KUKA KRL data list: Glode_HanGao.dat

&ACCESS RVO1
&REL 506
&PARAM EDITMASK = *
&PARAM TEMPLATE = C:\KRC\Roboter\Template\vorgabe
&PARAM DISKPATH = KRC:\R1\Program\HG
DEFDAT  GLODE_HANGAO PUBLIC



GLOBAL BOOL EKI_Server_Ini=TRUE
GLOBAL BOOL EKI_Server_Open=TRUE
GLOBAL BOOL EKI_Server_Connect=TRUE
GLOBAL BOOL EKI_Server_Receive=FALSE
GLOBAL BOOL EKI_Server_Send=FALSE
GLOBAL BOOL EKI_Server_Reset=FALSE


;--------DECL_Enum---------------
GLOBAL ENUM Sink_Type_Enum UpDown_One,LeftRight_One,LeftRight_Two,Null
GLOBAL ENUM Area_Enum L0,C45,L90,C135,L180,C225,L270,C315,N45,N135,N225,N315
GLOBAL ENUM Pos_Type_Enum C_LIN_POS,C_CIR_POS,L_LIN_POS
GLOBAL ENUM Work_Area_Enum A0,A90,A270
GLOBAL ENUM Vision_Model_Enum Calibration,Find_Model
GLOBAL ENUM Vision_Type_Enum Vision_Run,Vision_No,Vision_Text
GLOBAL ENUM Vision_PATH_Enum X,Y,Z,XY,XZ,YZ,XYZ,XYZABC
;----------------------------------
;---DECL-STRUC-------------------------


GLOBAL STRUC Surround_Welding_Type BOOL Write_Status,REAL Sink_Size_Long,REAL Sink_Size_Width,REAL Sink_Size_R,REAL Sink_Size_Short_Side,REAL Sink_Size_Short_OnePos,REAL Sink_Size_Short_TwoPos,REAL Sink_Size_Pots_Thick,REAL Sink_Size_Panel_Thick,INT Sink_Model,REAL Sink_Size_Left_Distance,REAL Sink_Size_Down_Distance,Sink_Type_Enum Sink_Type
GLOBAL STRUC LSC_TOOL_TYP INT LSR_MAX_PWR,INT LSR_MIN_PWR,INT LSR_Prg,REAL SNSR_Prg,INT SNSR_State,REAL GAS_Pressure,INT LSR_Dly,INT GAS_Pre_Flow,INT GAS_Post_Flow
GLOBAL STRUC Offset_POS REAL X,REAL Y,REAL Z,REAL A,REAL B,REAL C
GLOBAL STRUC Offset_CIR REAL C_X,REAL C_Y,REAL C_Z,REAL C_A,REAL C_B,REAL C_C
GLOBAL STRUC Calculate_Lin_Const REAL A,REAL B,REAL C
GLOBAL STRUC Calibration_Sink_TYP REAL Long,REAL Width
GLOBAL STRUC Calibrate_Data BOOL Calibrate_State,INT Plan_Base_No,CHAR Calib_Pos_Name_1[20],CHAR Calib_Pos_Name_2[20],CHAR Calib_Pos_Name_3[20],CHAR Calib_Pos_Name_4[20],CHAR Calib_Pos_Name_5[20],CHAR Calib_Pos_Name_6[20],CHAR Calib_Pos_Name_7[20],CHAR Calib_Pos_Name_8[20],CHAR Calib_Pos_Name_9[20],CHAR Calib_Pos_Name_10[20]



GLOBAL STRUC Surr_Welding_Craft_Type CHAR Welding_Name[20],E6POS Welding_Pos,REAL Welding_Power,REAL Welding_Speed,REAL Welding_Angle,INT Welding_CDIS,INT Welding_ACC,Offset_POS Welding_Offset,Offset_CIR Welding_Offset_CIR



;-------------------------------------


;----------DECL_Value----------------------
DECL GLOBAL Surround_Welding_Type SW_DEFAULT={Sink_Size_Long 50.0000,Sink_Size_Width 345.000,Sink_Size_R 10.0000,Sink_Size_Pots_Thick 0.750000,Sink_Size_Panel_Thick 2.85000,Sink_Model 952154,Sink_Type #UpDown_One}
DECL GLOBAL LSC_TOOL_TYP LTDEFAULT={LSR_MAX_PWR 500,LSR_MIN_PWR 50,LSR_Prg 1,SNSR_Prg 1.00000,SNSR_State 0,GAS_Pressure 1.00000,LSR_Dly 100,GAS_Pre_Flow 0,GAS_Post_Flow 0}
DECL GLOBAL Offset_POS FFDEFAULT={X 0.0,Y 0.0,Z 0.0,A 0.0,B 0.0,C 0.0}
DECL GLOBAL Offset_CIR FCDEFAULT={C_X 0.0,C_Y 0.0,C_Z 0.0,C_A 0.0,C_B 0.0,C_C 0.0}
DECL GLOBAL Calibrate_Data CDDEFAULT={Calibrate_State FALSE,Plan_Base_No 5,Calib_Pos_Name_1[] " ",Calib_Pos_Name_2[] " ",Calib_Pos_Name_3[] " ",Calib_Pos_Name_4[] " ",Calib_Pos_Name_5[] " ",Calib_Pos_Name_6[] " ",Calib_Pos_Name_7[] " ",Calib_Pos_Name_8[] " ",Calib_Pos_Name_9[] " ",Calib_Pos_Name_10[] " "}
DECL GLOBAL E6POS PODEFAULT={X 0.0,Y 0.0,Z 0.0,A 0.0,B 0.0,C 0.0}
DECL GLOBAL E6POS XDEFAULT={X 0.0,Y 0.0,Z 0.0,A 0.0,B 0.0,C 0.0,S 2,T 2,E1 0.0,E2 0.0,E3 0.0,E4 0.0,E5 0.0,E6 0.0}



DECL GLOBAL Surround_Welding_Type Camera_Calibration_Data={Sink_Size_Long 632.000,Sink_Size_Width 352.000,Sink_Size_R 10.0000,Sink_Size_Short_Side 23.0000,Sink_Size_Short_OnePos 36.0000,Sink_Size_Short_TwoPos 328.000,Sink_Size_Pots_Thick 0.0,Sink_Size_Panel_Thick 0.0,Sink_Model 952154,Sink_Size_Left_Distance 24.0000,Sink_Size_Down_Distance 24.0000,Sink_Type #LeftRight_One}

DECL GLOBAL E6POS N1_Cam_45_POS={X 293.000,Y 90.0000,Z -80.0000,A 0.0,B 0.0,C 0.0,S 2,T 10,E1 0.0,E2 0.0,E3 0.0,E4 0.0,E5 0.0,E6 0.0}
DECL GLOBAL E6POS N1_Cam_135_POS={X -42.0000,Y 90.0000,Z -80.0000,A 0.0,B 0.0,C 0.0,S 2,T 10,E1 0.0,E2 0.0,E3 0.0,E4 0.0,E5 0.0,E6 0.0}
DECL GLOBAL E6POS N1_Cam_225_POS={X -40.0000,Y 716.000,Z -80.0000,A 0.0,B 0.0,C 0.0,S 2,T 43,E1 0.0,E2 0.0,E3 0.0,E4 0.0,E5 0.0,E6 0.0}
DECL GLOBAL E6POS N1_Cam_315_POS={X 295.000,Y 714.000,Z -80.0000,A 0.0,B 0.0,C 0.0,S 2,T 43,E1 0.0,E2 0.0,E3 0.0,E4 0.0,E5 0.0,E6 0.0}

DECL GLOBAL E6POS N2_Cam_45_POS={X 293.122131,Y 89.9176636,Z -80.0293961,A 0.0,B 0.0,C 0.0,S 2,T 10,E1 0.0,E2 0.0,E3 0.0,E4 0.0,E5 0.0,E6 0.0}
DECL GLOBAL E6POS N2_Cam_135_POS={X -42.3839874,Y 91.8151550,Z -80.0254822,A 0.0,B 0.0,C 0.0,S 2,T 10,E1 0.0,E2 0.0,E3 0.0,E4 0.0,E5 0.0,E6 0.0}
DECL GLOBAL E6POS N2_Cam_225_POS={X -39.7999954,Y 716.082336,Z -80.0293350,A 0.0,B 0.0,C 0.0,S 2,T 43,E1 0.0,E2 0.0,E3 0.0,E4 0.0,E5 0.0,E6 0.0}
DECL GLOBAL E6POS N2_Cam_315_POS={X 294.984924,Y 714.198059,Z -80.0293350,A 0.0,B 0.0,C 0.0,S 2,T 43,E1 0.0,E2 0.0,E3 0.0,E4 0.0,E5 0.0,E6 0.0}

DECL GLOBAL E6POS N45_OFFSET_POS={X 375.888,Y 19.1080,Z 0.0,A 0.0,B 0.0,C 0.0}
DECL GLOBAL E6POS N135_OFFSET_POS={X 19.2480,Y 19.4280,Z 0.0,A 0.0,B 0.0,C 0.0}
DECL GLOBAL E6POS N225_OFFSET_POS={X 18.8370,Y 660.925,Z 0.0,A 0.0,B 0.0,C 0.0}
DECL GLOBAL E6POS N315_OFFSET_POS={X 375.531,Y 661.361,Z 0.0,A 0.0,B 0.0,C 0.0}

DECL GLOBAL E6POS N45_CIR_POS={X 370.887,Y 21.4200,Z 0.0,A 0.0,B 0.0,C 0.0}
DECL GLOBAL E6POS N135_CIR_POS={X 23.1220,Y 23.0800,Z 0.0,A 0.0,B 0.0,C 0.0}
DECL GLOBAL E6POS N225_CIR_POS={X 22.5580,Y 657.093,Z 0.0,A 0.0,B 0.0,C 0.0}
DECL GLOBAL E6POS N315_CIR_POS={X 371.252,Y 658.128,Z 0.0,A 0.0,B 0.0,C 0.0}

DECL GLOBAL E6POS D45_Start_POS={X 363.069,Y 0.172000,Z 0.0,A 0.0,B 0.0,C 0.0}
DECL GLOBAL E6POS D45_End_POS={X 363.226,Y 19.0740,Z 0.0,A 0.0,B 0.0,C 0.0}
DECL GLOBAL E6POS D135_Start_POS={X 31.9650,Y 0.265000,Z 0.0,A 0.0,B 0.0,C 0.0}
DECL GLOBAL E6POS D135_End_POS={X 31.7740,Y 19.3580,Z 0.0,A 0.0,B 0.0,C 0.0}
DECL GLOBAL E6POS D225_Start_POS={X 31.1060,Y 680.043,Z 0.0,A 0.0,B 0.0,C 0.0}
DECL GLOBAL E6POS D225_End_POS={X 30.9840,Y 660.897,Z 0.0,A 0.0,B 0.0,C 0.0}
DECL GLOBAL E6POS D315_Start_POS={X 363.308,Y 680.243,Z 0.0,A 0.0,B 0.0,C 0.0}
DECL GLOBAL E6POS D315_End_POS={X 363.008,Y 661.355,Z 0.0,A 0.0,B 0.0,C 0.0}


DECL GLOBAL Surr_Welding_Craft_Type L0_Welding_Craft[2,10]
L0_Welding_Craft[1,1]={Welding_Name[] "S2",Welding_Pos {X 375.389648,Y 92.3825073,Z 1.50000,A 0.0,B 20.0000,C 0.0},Welding_Power 58.0000,Welding_Speed 0.400000,Welding_Angle 20.0000,Welding_CDIS 5,Welding_ACC 100,Welding_Offset {X 0.0,Y 0.0,Z 0.0}}
L0_Welding_Craft[1,2]={Welding_Name[] "L0_S2",Welding_Pos {X 375.159363,Y 586.834473,Z 1.50000,A 0.0,B 20.0000,C 0.0},Welding_Power 58.0000,Welding_Speed 0.0450000,Welding_Angle 20.0000,Welding_CDIS 5,Welding_ACC 100,Welding_Offset {X -1.00000,Y 0.0,Z 0.0}}
L0_Welding_Craft[1,3]={Welding_Name[] "L0_S3",Welding_Pos {X 375.274506,Y 339.608490,Z 1.50000,A 0.0,B 20.0000,C 0.0},Welding_Power 58.0000,Welding_Speed 0.0450000,Welding_Angle 20.0000,Welding_CDIS 5,Welding_ACC 100,Welding_Offset {X -0.500000,Y 0.0,Z 0.0}}
L0_Welding_Craft[1,4]={Welding_Name[] "L0_S4",Welding_Pos {X 375.418427,Y 30.5759888,Z 1.50000,A 0.0,B 20.0000,C 0.0},Welding_Power 58.0000,Welding_Speed 0.0450000,Welding_Angle 20.0000,Welding_CDIS 5,Welding_ACC 100,Welding_Offset {X -0.500000,Y 0.0,Z 0.0}}
L0_Welding_Craft[1,5]={Welding_Name[] "S1",Welding_Pos {X 400.000,Y 86.0000153,Z -3.00000,A 0.0,B 23.0000,C 0.0},Welding_Power 80.0000,Welding_Speed 0.0400000,Welding_Angle 20.0000,Welding_CDIS 5,Welding_ACC 100,Welding_Offset {X 0.0,Y 0.0,Z 0.0}}
L0_Welding_Craft[1,6]={Welding_Name[] "S6",Welding_Pos {X 533.000,Y 463.600037,Z -2.05000,A 0.0,B -23.0000,C 0.0},Welding_Power 80.0000,Welding_Speed 0.0400000,Welding_Angle 20.0000,Welding_CDIS 5,Welding_ACC 100,Welding_Offset {X 0.0,Y 0.0,Z 0.0}}
L0_Welding_Craft[1,7]={Welding_Name[] "S7",Welding_Pos {X 533.000,Y 463.600037,Z -2.05000,A 0.0,B -23.0000,C 0.0},Welding_Power 80.0000,Welding_Speed 0.0400000,Welding_Angle 20.0000,Welding_CDIS 5,Welding_ACC 100,Welding_Offset {X 0.0,Y 0.0,Z 0.0}}
L0_Welding_Craft[1,8]={Welding_Name[] "S8",Welding_Pos {X 533.000,Y 463.600037,Z -2.05000,A 0.0,B -23.0000,C 0.0},Welding_Power 80.0000,Welding_Speed 0.0400000,Welding_Angle 20.0000,Welding_CDIS 5,Welding_ACC 100,Welding_Offset {X 0.0,Y 0.0,Z 0.0}}
L0_Welding_Craft[1,9]={Welding_Name[] "S9",Welding_Pos {X 533.000,Y 463.600037,Z -2.05000,A 0.0,B -23.0000,C 0.0},Welding_Power 80.0000,Welding_Speed 0.0400000,Welding_Angle 20.0000,Welding_CDIS 5,Welding_ACC 100,Welding_Offset {X 0.0,Y 0.0,Z 0.0}}
L0_Welding_Craft[1,10]={Welding_Name[] "S10",Welding_Pos {X 533.000,Y 338.000,Z -2.05000,A 0.0,B -23.0000,C 0.0},Welding_Power 80.0000,Welding_Speed 0.0400000,Welding_Angle 20.0000,Welding_CDIS 5,Welding_ACC 100,Welding_Offset {X 0.0,Y 0.0,Z 0.0}}
L0_Welding_Craft[2,1]={Welding_Name[] "L0_S1",Welding_Pos {X 375.846954,Y 92.9332886,Z 1.50000,A 0.0,B 20.0000,C 0.0},Welding_Power 60.0000,Welding_Speed 0.480000,Welding_Angle 20.0000,Welding_CDIS 0,Welding_ACC 100,Welding_Offset {X 0.100000,Y 0.0,Z 1.00000}}
L0_Welding_Craft[2,2]={Welding_Name[] "L0_S2",Welding_Pos {X 375.572052,Y 587.535706,Z 1.50000,A 0.0,B 20.0000,C 0.0},Welding_Power 60.0000,Welding_Speed 0.0450000,Welding_Angle 20.0000,Welding_CDIS 5,Welding_ACC 100,Welding_Offset {X -0.200000,Y 0.0,Z 1.00000}}
L0_Welding_Craft[2,3]={Welding_Name[] "L0_S3",Welding_Pos {X 375.709503,Y 340.234497,Z 1.50000,A 0.0,B 20.0000,C 0.0},Welding_Power 60.0000,Welding_Speed 0.0450000,Welding_Angle 20.0000,Welding_CDIS 5,Welding_ACC 100,Welding_Offset {X -0.300000,Y 0.0,Z 1.00000}}
L0_Welding_Craft[2,4]={Welding_Name[] "L0_S4",Welding_Pos {X 375.881317,Y 31.1079712,Z 1.50000,A 0.0,B 20.0000,C 0.0},Welding_Power 60.0000,Welding_Speed 0.0400000,Welding_Angle 20.0000,Welding_CDIS 5,Welding_ACC 100,Welding_Offset {X -0.200000,Y 0.0,Z 1.00000}}
L0_Welding_Craft[2,5]={Welding_Name[] "S1",Welding_Pos {X 400.000,Y 86.0000153,Z -3.00000,A 0.0,B 23.0000,C 0.0},Welding_Power 80.0000,Welding_Speed 0.0400000,Welding_Angle 20.0000,Welding_CDIS 5,Welding_ACC 100,Welding_Offset {X 0.0,Y 0.0,Z 0.0}}
L0_Welding_Craft[2,6]={Welding_Name[] "S6",Welding_Pos {X 533.000,Y 463.600037,Z -2.05000,A 0.0,B -23.0000,C 0.0},Welding_Power 80.0000,Welding_Speed 0.0400000,Welding_Angle 20.0000,Welding_CDIS 5,Welding_ACC 100,Welding_Offset {X 0.0,Y 0.0,Z 0.0}}
L0_Welding_Craft[2,7]={Welding_Name[] "S7",Welding_Pos {X 533.000,Y 463.600037,Z -2.05000,A 0.0,B -23.0000,C 0.0},Welding_Power 80.0000,Welding_Speed 0.0400000,Welding_Angle 20.0000,Welding_CDIS 5,Welding_ACC 100,Welding_Offset {X 0.0,Y 0.0,Z 0.0}}
L0_Welding_Craft[2,8]={Welding_Name[] "S8",Welding_Pos {X 533.000,Y 463.600037,Z -2.05000,A 0.0,B -23.0000,C 0.0},Welding_Power 80.0000,Welding_Speed 0.0400000,Welding_Angle 20.0000,Welding_CDIS 5,Welding_ACC 100,Welding_Offset {X 0.0,Y 0.0,Z 0.0}}
L0_Welding_Craft[2,9]={Welding_Name[] "S9",Welding_Pos {X 533.000,Y 463.600037,Z -2.05000,A 0.0,B -23.0000,C 0.0},Welding_Power 80.0000,Welding_Speed 0.0400000,Welding_Angle 20.0000,Welding_CDIS 5,Welding_ACC 100,Welding_Offset {X 0.0,Y 0.0,Z 0.0}}
L0_Welding_Craft[2,10]={Welding_Name[] "S10",Welding_Pos {X 533.000,Y 338.000,Z -2.05000,A 0.0,B -23.0000,C 0.0},Welding_Power 80.0000,Welding_Speed 0.0400000,Welding_Angle 20.0000,Welding_CDIS 5,Welding_ACC 100,Welding_Offset {X 0.0,Y 0.0,Z 0.0}}



DECL GLOBAL Surr_Welding_Craft_Type C45_Welding_Craft[2,3]
C45_Welding_Craft[1,1]={Welding_Name[] "C45_S1",Welding_Pos {X 375.418427,Y 30.5759888,Z 1.50000,A 0.0,B 20.0000,C 0.0},Welding_Power 80.0000,Welding_Speed 0.0400000,Welding_Angle 20.0000,Welding_CDIS 5,Welding_ACC 100,Welding_Offset {X 0.0,Y 0.0,Z -1.00000}}
C45_Welding_Craft[1,2]={Welding_Name[] "PM3",Welding_Pos {X 370.291,Y 20.8820,Z 1.50000,A 0.0,B 0.0,C 0.0},Welding_Power 80.0000,Welding_Speed 0.0400000,Welding_Angle 20.0000,Welding_CDIS 5,Welding_ACC 100,Welding_Offset {X 0.500000,Y 0.500000,Z -1.00000},Welding_Offset_CIR {C_X 0.0,C_Y 0.0,C_Z 0.0}}
C45_Welding_Craft[1,3]={Welding_Name[] "PE3",Welding_Pos {X 363.424,Y 18.5840397,Z 1.50000,A 0.0,B 0.0,C 20.0000},Welding_Power 58.0000,Welding_Speed 0.0200000,Welding_Angle 20.0000,Welding_CDIS 5,Welding_ACC 100,Welding_Offset {X 0.0,Y 0.0,Z -1.00000}}
C45_Welding_Craft[2,1]={Welding_Name[] "C45_S1",Welding_Pos {X 375.881317,Y 31.1079712,Z 1.50000,A 0.0,B 20.0000,C 0.0},Welding_Power 65.0000,Welding_Speed 0.0400000,Welding_Angle 20.0000,Welding_CDIS 40,Welding_ACC 80,Welding_Offset {X 0.0,Y 0.0,Z 0.0}}
C45_Welding_Craft[2,2]={Welding_Name[] "PM3",Welding_Pos {X 370.887,Y 21.4200,Z 1.50000,A 0.0,B 0.0,C 0.0},Welding_Power 60.0000,Welding_Speed 0.0400000,Welding_Angle 20.0000,Welding_CDIS 5,Welding_ACC 100,Welding_Offset {X 1.60000,Y 2.30000,Z 0.0},Welding_Offset_CIR {C_X 0.0,C_Y 0.0,C_Z 0.0}}
C45_Welding_Craft[2,3]={Welding_Name[] "PE3",Welding_Pos {X 363.888,Y 19.1187668,Z 1.50000,A 0.0,B 0.0,C 20.0000},Welding_Power 60.0000,Welding_Speed 0.0230000,Welding_Angle 20.0000,Welding_CDIS 5,Welding_ACC 100,Welding_Offset {X 0.0,Y 0.200000,Z 0.0}}


DECL GLOBAL Surr_Welding_Craft_Type L90_Welding_Craft[2,10]
L90_Welding_Craft[1,1]={Welding_Name[] "L90_S1",Welding_Pos {X 330.151611,Y 18.6063309,Z 1.50000,A 0.0,B 0.0,C 20.0000},Welding_Power 58.0000,Welding_Speed 0.0400000,Welding_Angle 20.0000,Welding_CDIS 5,Welding_ACC 100,Welding_Offset {X 0.0,Y 0.0,Z 0.0}}
L90_Welding_Craft[1,2]={Welding_Name[] "L90_S2",Welding_Pos {X 197.062012,Y 18.6955,Z 1.50000,A 0.0,B 0.0,C 20.0000},Welding_Power 58.0000,Welding_Speed 0.0400000,Welding_Angle 20.0000,Welding_CDIS 5,Welding_ACC 100,Welding_Offset {X 0.0,Y 0.0,Z 0.0}}
L90_Welding_Craft[1,3]={Welding_Name[] "L90_S3",Welding_Pos {X 63.9724121,Y 18.7846680,Z 1.50000,A 0.0,B 0.0,C 20.0000},Welding_Power 58.0000,Welding_Speed 0.0400000,Welding_Angle 20.0000,Welding_CDIS 5,Welding_ACC 100,Welding_Offset {X 0.0,Y -0.500000,Z 0.0}}
L90_Welding_Craft[1,4]={Welding_Name[] "S4",Welding_Pos {X 400.000,Y 86.0000153,Z -3.00000,A 0.0,B 23.0000,C 0.0},Welding_Power 80.0000,Welding_Speed 0.0400000,Welding_Angle 20.0000,Welding_CDIS 5,Welding_ACC 100,Welding_Offset {X 0.0,Y 0.0,Z 0.0}}
L90_Welding_Craft[1,5]={Welding_Name[] "S5",Welding_Pos {X 371.000,Y 0.0,Z -3.00000,A 0.0,B 0.0,C 23.0000},Welding_Power 80.0000,Welding_Speed 0.0400000,Welding_Angle 20.0000,Welding_CDIS 5,Welding_ACC 100,Welding_Offset {X 0.0,Y 0.0,Z 0.0}}
L90_Welding_Craft[1,6]={Welding_Name[] "S6",Welding_Pos {X 533.000,Y 463.600037,Z -2.05000,A 0.0,B -23.0000,C 0.0},Welding_Power 80.0000,Welding_Speed 0.0400000,Welding_Angle 20.0000,Welding_CDIS 5,Welding_ACC 100,Welding_Offset {X 0.0,Y 0.0,Z 0.0}}
L90_Welding_Craft[1,7]={Welding_Name[] "S7",Welding_Pos {X 533.000,Y 463.600037,Z -2.05000,A 0.0,B -23.0000,C 0.0},Welding_Power 80.0000,Welding_Speed 0.0400000,Welding_Angle 20.0000,Welding_CDIS 5,Welding_ACC 100,Welding_Offset {X 0.0,Y 0.0,Z 0.0}}
L90_Welding_Craft[1,8]={Welding_Name[] "S8",Welding_Pos {X 533.000,Y 463.600037,Z -2.05000,A 0.0,B -23.0000,C 0.0},Welding_Power 80.0000,Welding_Speed 0.0400000,Welding_Angle 20.0000,Welding_CDIS 5,Welding_ACC 100,Welding_Offset {X 0.0,Y 0.0,Z 0.0}}
L90_Welding_Craft[1,9]={Welding_Name[] "S9",Welding_Pos {X 533.000,Y 463.600037,Z -2.05000,A 0.0,B -23.0000,C 0.0},Welding_Power 80.0000,Welding_Speed 0.0400000,Welding_Angle 20.0000,Welding_CDIS 5,Welding_ACC 100,Welding_Offset {X 0.0,Y 0.0,Z 0.0}}
L90_Welding_Craft[1,10]={Welding_Name[] "S10",Welding_Pos {X 533.000,Y 338.000,Z -2.05000,A 0.0,B -23.0000,C 0.0},Welding_Power 80.0000,Welding_Speed 0.0400000,Welding_Angle 20.0000,Welding_CDIS 5,Welding_ACC 100,Welding_Offset {X 0.0,Y 0.0,Z 0.0}}
L90_Welding_Craft[2,1]={Welding_Name[] "L90_S1",Welding_Pos {X 330.624,Y 19.1486130,Z 1.50000,A 0.0,B 0.0,C 20.0000},Welding_Power 63.0000,Welding_Speed 0.0450000,Welding_Angle 20.0000,Welding_CDIS 5,Welding_ACC 100,Welding_Offset {X 0.0,Y 0.400000,Z 0.0}}
L90_Welding_Craft[2,2]={Welding_Name[] "L90_S2",Welding_Pos {X 197.568,Y 19.2680,Z 1.50000,A 0.0,B 0.0,C 20.0000},Welding_Power 63.0000,Welding_Speed 0.0450000,Welding_Angle 20.0000,Welding_CDIS 5,Welding_ACC 100,Welding_Offset {X 0.0,Y 0.0,Z 0.0}}
L90_Welding_Craft[2,3]={Welding_Name[] "L90_S3",Welding_Pos {X 64.5119934,Y 19.3873863,Z 1.50000,A 0.0,B 0.0,C 20.0000},Welding_Power 60.0000,Welding_Speed 0.0450000,Welding_Angle 20.0000,Welding_CDIS 5,Welding_ACC 100,Welding_Offset {X 0.0,Y -0.400000,Z 0.0}}
L90_Welding_Craft[2,4]={Welding_Name[] "S4",Welding_Pos {X 400.000,Y 86.0000153,Z -3.00000,A 0.0,B 23.0000,C 0.0},Welding_Power 80.0000,Welding_Speed 0.0430000,Welding_Angle 20.0000,Welding_CDIS 5,Welding_ACC 100,Welding_Offset {X 0.0,Y 0.0,Z 0.0}}
L90_Welding_Craft[2,5]={Welding_Name[] "S5",Welding_Pos {X 371.000,Y 0.0,Z -3.00000,A 0.0,B 0.0,C 23.0000},Welding_Power 80.0000,Welding_Speed 0.0400000,Welding_Angle 20.0000,Welding_CDIS 5,Welding_ACC 100,Welding_Offset {X 0.0,Y 0.0,Z 0.0}}
L90_Welding_Craft[2,6]={Welding_Name[] "S6",Welding_Pos {X 533.000,Y 463.600037,Z -2.05000,A 0.0,B -23.0000,C 0.0},Welding_Power 80.0000,Welding_Speed 0.0400000,Welding_Angle 20.0000,Welding_CDIS 5,Welding_ACC 100,Welding_Offset {X 0.0,Y 0.0,Z 0.0}}
L90_Welding_Craft[2,7]={Welding_Name[] "S7",Welding_Pos {X 533.000,Y 463.600037,Z -2.05000,A 0.0,B -23.0000,C 0.0},Welding_Power 80.0000,Welding_Speed 0.0400000,Welding_Angle 20.0000,Welding_CDIS 5,Welding_ACC 100,Welding_Offset {X 0.0,Y 0.0,Z 0.0}}
L90_Welding_Craft[2,8]={Welding_Name[] "S8",Welding_Pos {X 533.000,Y 463.600037,Z -2.05000,A 0.0,B -23.0000,C 0.0},Welding_Power 80.0000,Welding_Speed 0.0400000,Welding_Angle 20.0000,Welding_CDIS 5,Welding_ACC 100,Welding_Offset {X 0.0,Y 0.0,Z 0.0}}
L90_Welding_Craft[2,9]={Welding_Name[] "S9",Welding_Pos {X 533.000,Y 463.600037,Z -2.05000,A 0.0,B -23.0000,C 0.0},Welding_Power 80.0000,Welding_Speed 0.0400000,Welding_Angle 20.0000,Welding_CDIS 5,Welding_ACC 100,Welding_Offset {X 0.0,Y 0.0,Z 0.0}}
L90_Welding_Craft[2,10]={Welding_Name[] "S10",Welding_Pos {X 533.000,Y 338.000,Z -2.05000,A 0.0,B -23.0000,C 0.0},Welding_Power 80.0000,Welding_Speed 0.0400000,Welding_Angle 20.0000,Welding_CDIS 5,Welding_ACC 100,Welding_Offset {X 0.0,Y 0.0,Z 0.0}}

DECL GLOBAL Surr_Welding_Craft_Type C135_Welding_Craft[2,3]
C135_Welding_Craft[1,1]={Welding_Name[] "C135_S1",Welding_Pos {X 30.7000122,Y 18.8069611,Z 1.50000,A 0.0,B 0.0,C 20.0000},Welding_Power 80.0000,Welding_Speed 0.0400000,Welding_Angle 20.0000,Welding_CDIS 5,Welding_ACC 100,Welding_Offset {X 0.0,Y -0.500000,Z -1.00000}}
C135_Welding_Craft[1,2]={Welding_Name[] "PM4",Welding_Pos {X 21.8080,Y 22.4770,Z 1.50000,A 0.0,B 0.0,C 0.0},Welding_Power 80.0000,Welding_Speed 0.0400000,Welding_Angle -20.0000,Welding_CDIS 5,Welding_ACC 100,Welding_Offset {X -0.500000,Y -0.500000,Z -1.00000},Welding_Offset_CIR {C_X 0.0,C_Y 0.0,C_Z 0.0}}
C135_Welding_Craft[1,3]={Welding_Name[] "PE4",Welding_Pos {X 18.6979065,Y 30.8150,Z 1.50000,A 0.0,B -20.0000,C 0.0},Welding_Power 58.0000,Welding_Speed 0.0200000,Welding_Angle -20.0000,Welding_CDIS 5,Welding_ACC 100,Welding_Offset {X -0.500000,Y 0.0,Z -1.00000}}
C135_Welding_Craft[2,1]={Welding_Name[] "C135_S1",Welding_Pos {X 31.2479858,Y 19.4172325,Z 1.50000,A 0.0,B 0.0,C 20.0000},Welding_Power 60.0000,Welding_Speed 0.0400000,Welding_Angle 20.0000,Welding_CDIS 5,Welding_ACC 100,Welding_Offset {X 0.0,Y -0.300000,Z 0.0}}
C135_Welding_Craft[2,2]={Welding_Name[] "PM4",Welding_Pos {X 23.1220,Y 23.0800,Z 1.50000,A 0.0,B 0.0,C 0.0},Welding_Power 60.0000,Welding_Speed 0.0400000,Welding_Angle -20.0000,Welding_CDIS 5,Welding_ACC 100,Welding_Offset {X 0.0,Y -1.40000,Z 0.0},Welding_Offset_CIR {C_X 0.0,C_Y 0.0,C_Z 0.0}}
C135_Welding_Craft[2,3]={Welding_Name[] "PE4",Welding_Pos {X 19.2403107,Y 31.4279976,Z 1.50000,A 0.0,B -20.0000,C 0.0},Welding_Power 60.0000,Welding_Speed 0.0200000,Welding_Angle -20.0000,Welding_CDIS 5,Welding_ACC 100,Welding_Offset {X -0.500000,Y -0.300000,Z 0.0}}

DECL GLOBAL Surr_Welding_Craft_Type L180_Welding_Craft[2,10]
L180_Welding_Craft[1,1]={Welding_Name[] "L180_S1",Welding_Pos {X 18.6871262,Y 92.5788956,Z 1.50000,A 0.0,B -20.0000,C 0.0},Welding_Power 58.0000,Welding_Speed 0.0400000,Welding_Angle -20.0000,Welding_CDIS 5,Welding_ACC 100,Welding_Offset {X -0.500000,Y 0.0,Z 0.0}}
L180_Welding_Craft[1,2]={Welding_Name[] "L180_S2",Welding_Pos {X 18.6440010,Y 339.634491,Z 1.50000,A 0.0,B -20.0000,C 0.0},Welding_Power 58.0000,Welding_Speed 0.0400000,Welding_Angle -20.0000,Welding_CDIS 5,Welding_ACC 100,Welding_Offset {X -0.200000,Y 2.77555756E-17,Z 0.0}}
L180_Welding_Craft[1,3]={Welding_Name[] "L180_S3",Welding_Pos {X 18.5954838,Y 617.572,Z 1.50000,A 0.0,B -20.0000,C 0.0},Welding_Power 58.0000,Welding_Speed 0.0400000,Welding_Angle -20.0000,Welding_CDIS 5,Welding_ACC 100,Welding_Offset {X 0.0,Y 0.0,Z 0.0}}
L180_Welding_Craft[1,4]={Welding_Name[] "S4",Welding_Pos {X 400.000,Y 86.0000153,Z -3.00000,A 0.0,B 23.0000,C 0.0},Welding_Power 80.0000,Welding_Speed 0.0400000,Welding_Angle -20.0000,Welding_CDIS 5,Welding_ACC 100,Welding_Offset {X 0.0,Y 0.0,Z 0.0}}
L180_Welding_Craft[1,5]={Welding_Name[] "S5",Welding_Pos {X 0.0,Y 371.000,Z -3.00000,A 0.0,B -23.0000,C 0.0},Welding_Power 80.0000,Welding_Speed 0.0400000,Welding_Angle -20.0000,Welding_CDIS 5,Welding_ACC 100,Welding_Offset {X 0.0,Y 0.0,Z 0.0}}
L180_Welding_Craft[1,6]={Welding_Name[] "S6",Welding_Pos {X 533.000,Y 463.600037,Z -2.05000,A 0.0,B -23.0000,C 0.0},Welding_Power 80.0000,Welding_Speed 0.0400000,Welding_Angle -20.0000,Welding_CDIS 5,Welding_ACC 100,Welding_Offset {X 0.0,Y 0.0,Z 0.0}}
L180_Welding_Craft[1,7]={Welding_Name[] "S7",Welding_Pos {X 533.000,Y 463.600037,Z -2.05000,A 0.0,B -23.0000,C 0.0},Welding_Power 80.0000,Welding_Speed 0.0400000,Welding_Angle -20.0000,Welding_CDIS 5,Welding_ACC 100,Welding_Offset {X 0.0,Y 0.0,Z 0.0}}
L180_Welding_Craft[1,8]={Welding_Name[] "S8",Welding_Pos {X 533.000,Y 463.600037,Z -2.05000,A 0.0,B -23.0000,C 0.0},Welding_Power 80.0000,Welding_Speed 0.0400000,Welding_Angle -20.0000,Welding_CDIS 5,Welding_ACC 100,Welding_Offset {X 0.0,Y 0.0,Z 0.0}}
L180_Welding_Craft[1,9]={Welding_Name[] "S9",Welding_Pos {X 533.000,Y 463.600037,Z -2.05000,A 0.0,B -23.0000,C 0.0},Welding_Power 80.0000,Welding_Speed 0.0400000,Welding_Angle -20.0000,Welding_CDIS 5,Welding_ACC 100,Welding_Offset {X 0.0,Y 0.0,Z 0.0}}
L180_Welding_Craft[1,10]={Welding_Name[] "S10",Welding_Pos {X 533.000,Y 338.000,Z -2.05000,A 0.0,B -23.0000,C 0.0},Welding_Power 80.0000,Welding_Speed 0.0400000,Welding_Angle -20.0000,Welding_CDIS 5,Welding_ACC 100,Welding_Offset {X 0.0,Y 0.0,Z 0.0}}
L180_Welding_Craft[2,1]={Welding_Name[] "L180_S1",Welding_Pos {X 19.2007484,Y 93.1777,Z 1.50000,A 0.0,B -20.0000,C 0.0},Welding_Power 63.0000,Welding_Speed 0.0450000,Welding_Angle -20.0000,Welding_CDIS 5,Welding_ACC 100,Welding_Offset {X -0.700000,Y 0.0,Z 0.0}}
L180_Welding_Craft[2,2]={Welding_Name[] "L180_S2",Welding_Pos {X 19.0425,Y 340.176514,Z 1.50000,A 0.0,B -20.0000,C 0.0},Welding_Power 63.0000,Welding_Speed 0.0450000,Welding_Angle -20.0000,Welding_CDIS 5,Welding_ACC 100,Welding_Offset {X -0.300000,Y 0.0,Z 0.0}}
L180_Welding_Craft[2,3]={Welding_Name[] "L180_S3",Welding_Pos {X 18.8644695,Y 618.050110,Z 1.50000,A 0.0,B -20.0000,C 0.0},Welding_Power 63.0000,Welding_Speed 0.0450000,Welding_Angle -20.0000,Welding_CDIS 5,Welding_ACC 100,Welding_Offset {X -0.500000,Y 0.0,Z 0.0}}
L180_Welding_Craft[2,4]={Welding_Name[] "S4",Welding_Pos {X 400.000,Y 86.0000153,Z -3.00000,A 0.0,B 23.0000,C 0.0},Welding_Power 75.0000,Welding_Speed 0.0400000,Welding_Angle -20.0000,Welding_CDIS 5,Welding_ACC 100,Welding_Offset {X 0.0,Y 0.0,Z 0.0}}
L180_Welding_Craft[2,5]={Welding_Name[] "S5",Welding_Pos {X 0.0,Y 371.000,Z -3.00000,A 0.0,B -23.0000,C 0.0},Welding_Power 80.0000,Welding_Speed 0.0400000,Welding_Angle -20.0000,Welding_CDIS 5,Welding_ACC 100,Welding_Offset {X 0.0,Y 0.0,Z 0.0}}
L180_Welding_Craft[2,6]={Welding_Name[] "S6",Welding_Pos {X 533.000,Y 463.600037,Z -2.05000,A 0.0,B -23.0000,C 0.0},Welding_Power 80.0000,Welding_Speed 0.0400000,Welding_Angle -20.0000,Welding_CDIS 5,Welding_ACC 100,Welding_Offset {X 0.0,Y 0.0,Z 0.0}}
L180_Welding_Craft[2,7]={Welding_Name[] "S7",Welding_Pos {X 533.000,Y 463.600037,Z -2.05000,A 0.0,B -23.0000,C 0.0},Welding_Power 80.0000,Welding_Speed 0.0400000,Welding_Angle -20.0000,Welding_CDIS 5,Welding_ACC 100,Welding_Offset {X 0.0,Y 0.0,Z 0.0}}
L180_Welding_Craft[2,8]={Welding_Name[] "S8",Welding_Pos {X 533.000,Y 463.600037,Z -2.05000,A 0.0,B -23.0000,C 0.0},Welding_Power 80.0000,Welding_Speed 0.0400000,Welding_Angle -20.0000,Welding_CDIS 5,Welding_ACC 100,Welding_Offset {X 0.0,Y 0.0,Z 0.0}}
L180_Welding_Craft[2,9]={Welding_Name[] "S9",Welding_Pos {X 533.000,Y 463.600037,Z -2.05000,A 0.0,B -23.0000,C 0.0},Welding_Power 80.0000,Welding_Speed 0.0400000,Welding_Angle -20.0000,Welding_CDIS 5,Welding_ACC 100,Welding_Offset {X 0.0,Y 0.0,Z 0.0}}
L180_Welding_Craft[2,10]={Welding_Name[] "S10",Welding_Pos {X 533.000,Y 338.000,Z -2.05000,A 0.0,B -23.0000,C 0.0},Welding_Power 80.0000,Welding_Speed 0.0400000,Welding_Angle -20.0000,Welding_CDIS 5,Welding_ACC 100,Welding_Offset {X 0.0,Y 0.0,Z 0.0}}

DECL GLOBAL Surr_Welding_Craft_Type C225_Welding_Craft[2,3]
C225_Welding_Craft[1,1]={Welding_Name[] "C225_S1",Welding_Pos {X 18.5900936,Y 648.454,Z 1.50000,A 0.0,B -20.0000,C 0.0},Welding_Power 80.0000,Welding_Speed 0.0400000,Welding_Angle -20.0000,Welding_CDIS 5,Welding_ACC 100,Welding_Offset {X 0.0,Y 0.0,Z -1.00000}}
C225_Welding_Craft[1,2]={Welding_Name[] "PM5",Welding_Pos {X 22.1170,Y 656.630,Z 1.50000,A 0.0,B 0.0,C 0.0},Welding_Power 80.0000,Welding_Speed 0.0400000,Welding_Angle -20.0000,Welding_CDIS 5,Welding_ACC 100,Welding_Offset {X 0.500000,Y 0.500000,Z -1.00000},Welding_Offset_CIR {C_X 0.0,C_Y 0.0,C_Z 0.0}}
C225_Welding_Craft[1,3]={Welding_Name[] "PE5",Welding_Pos {X 30.5879974,Y 660.460266,Z 1.50000,A 0.0,B 0.0,C -20.0000},Welding_Power 58.0000,Welding_Speed 0.0200000,Welding_Angle -20.0000,Welding_CDIS 5,Welding_ACC 100,Welding_Offset {X 0.0,Y 0.0,Z -1.00000}}
C225_Welding_Craft[2,1]={Welding_Name[] "C225_S1",Welding_Pos {X 18.8446884,Y 648.925,Z 1.50000,A 0.0,B -20.0000,C 0.0},Welding_Power 60.0000,Welding_Speed 0.0430000,Welding_Angle -20.0000,Welding_CDIS 5,Welding_ACC 100,Welding_Offset {X -0.200000,Y 0.0,Z 0.0}}
C225_Welding_Craft[2,2]={Welding_Name[] "PM5",Welding_Pos {X 22.5580,Y 657.093,Z 1.50000,A 0.0,B 0.0,C 0.0},Welding_Power 60.0000,Welding_Speed 0.0400000,Welding_Angle -20.0000,Welding_CDIS 5,Welding_ACC 100,Welding_Offset {X 0.0,Y 0.700000,Z 0.0},Welding_Offset_CIR {C_X 0.0,C_Y 0.0,C_Z 0.0}}
C225_Welding_Craft[2,3]={Welding_Name[] "PE5",Welding_Pos {X 30.8369904,Y 660.939636,Z 1.50000,A 0.0,B 0.0,C -20.0000},Welding_Power 60.0000,Welding_Speed 0.0200000,Welding_Angle -20.0000,Welding_CDIS 5,Welding_ACC 100,Welding_Offset {X 0.0,Y 0.0,Z -1.00000}}

DECL GLOBAL Surr_Welding_Craft_Type L270_Welding_Craft[2,10]
L270_Welding_Craft[1,1]={Welding_Name[] "L270_S1",Welding_Pos {X 63.8416977,Y 660.477722,Z 1.50000,A 0.0,B 0.0,C -20.0000},Welding_Power 58.0000,Welding_Speed 0.0400000,Welding_Angle -20.0000,Welding_CDIS 5,Welding_ACC 100,Welding_Offset {X 0.0,Y 0.0,Z 0.0}}
L270_Welding_Craft[1,2]={Welding_Name[] "L270_S2",Welding_Pos {X 196.856491,Y 660.547485,Z 1.50000,A 0.0,B 0.0,C -20.0000},Welding_Power 58.0000,Welding_Speed 0.0400000,Welding_Angle -20.0000,Welding_CDIS 5,Welding_ACC 100,Welding_Offset {X 0.0,Y -0.300000,Z 0.0}}
L270_Welding_Craft[1,3]={Welding_Name[] "L270_S3",Welding_Pos {X 346.498108,Y 660.626,Z 1.50000,A 0.0,B 0.0,C -20.0000},Welding_Power 58.0000,Welding_Speed 0.0400000,Welding_Angle -20.0000,Welding_CDIS 5,Welding_ACC 100,Welding_Offset {X 0.0,Y -0.500000,Z 0.0}}
L270_Welding_Craft[1,4]={Welding_Name[] "S4",Welding_Pos {X 400.000,Y 86.0000153,Z -3.00000,A 0.0,B 23.0000,C 0.0},Welding_Power 80.0000,Welding_Speed 0.0400000,Welding_Angle -20.0000,Welding_CDIS 5,Welding_ACC 100,Welding_Offset {X 0.0,Y 0.0,Z 0.0}}
L270_Welding_Craft[1,5]={Welding_Name[] "S12",Welding_Pos {X 28.9999981,Y 400.000,Z -3.00000,A 0.0,B 0.0,C -23.0000},Welding_Power 80.0000,Welding_Speed 0.0400000,Welding_Angle -20.0000,Welding_CDIS 5,Welding_ACC 100,Welding_Offset {X 0.0,Y 0.0,Z 0.0}}
L270_Welding_Craft[1,6]={Welding_Name[] "S6",Welding_Pos {X 533.000,Y 463.600037,Z -2.05000,A 0.0,B -23.0000,C 0.0},Welding_Power 80.0000,Welding_Speed 0.0400000,Welding_Angle -20.0000,Welding_CDIS 5,Welding_ACC 100,Welding_Offset {X 0.0,Y 0.0,Z 0.0}}
L270_Welding_Craft[1,7]={Welding_Name[] "S7",Welding_Pos {X 533.000,Y 463.600037,Z -2.05000,A 0.0,B -23.0000,C 0.0},Welding_Power 80.0000,Welding_Speed 0.0400000,Welding_Angle -20.0000,Welding_CDIS 5,Welding_ACC 100,Welding_Offset {X 0.0,Y 0.0,Z 0.0}}
L270_Welding_Craft[1,8]={Welding_Name[] "S8",Welding_Pos {X 533.000,Y 463.600037,Z -2.05000,A 0.0,B -23.0000,C 0.0},Welding_Power 80.0000,Welding_Speed 0.0400000,Welding_Angle -20.0000,Welding_CDIS 5,Welding_ACC 100,Welding_Offset {X 0.0,Y 0.0,Z 0.0}}
L270_Welding_Craft[1,9]={Welding_Name[] "S9",Welding_Pos {X 533.000,Y 463.600037,Z -2.05000,A 0.0,B -23.0000,C 0.0},Welding_Power 80.0000,Welding_Speed 0.0400000,Welding_Angle -20.0000,Welding_CDIS 5,Welding_ACC 100,Welding_Offset {X 0.0,Y 0.0,Z 0.0}}
L270_Welding_Craft[1,10]={Welding_Name[] "S10",Welding_Pos {X 533.000,Y 338.000,Z -2.05000,A 0.0,B -23.0000,C 0.0},Welding_Power 80.0000,Welding_Speed 0.0400000,Welding_Angle -20.0000,Welding_CDIS 5,Welding_ACC 100,Welding_Offset {X 0.0,Y 0.0,Z 0.0}}
L270_Welding_Craft[2,1]={Welding_Name[] "L270_S1",Welding_Pos {X 64.1063919,Y 660.980286,Z 1.50000,A 0.0,B 0.0,C -20.0000},Welding_Power 60.0000,Welding_Speed 0.0450000,Welding_Angle -20.0000,Welding_CDIS 5,Welding_ACC 100,Welding_Offset {X 0.0,Y -0.100000,Z -1.00000}}
L270_Welding_Craft[2,2]={Welding_Name[] "L270_S2",Welding_Pos {X 197.184,Y 661.143,Z 1.50000,A 0.0,B 0.0,C -20.0000},Welding_Power 60.0000,Welding_Speed 0.0450000,Welding_Angle -20.0000,Welding_CDIS 5,Welding_ACC 100,Welding_Offset {X 0.0,Y -0.300000,Z 0.0}}
L270_Welding_Craft[2,3]={Welding_Name[] "L270_S3",Welding_Pos {X 346.896301,Y 661.326050,Z 1.50000,A 0.0,B 0.0,C -20.0000},Welding_Power 60.0000,Welding_Speed 0.0450000,Welding_Angle -20.0000,Welding_CDIS 5,Welding_ACC 100,Welding_Offset {X 0.0,Y -0.400000,Z 0.0}}
L270_Welding_Craft[2,4]={Welding_Name[] "S4",Welding_Pos {X 400.000,Y 86.0000153,Z -3.00000,A 0.0,B 23.0000,C 0.0},Welding_Power 80.0000,Welding_Speed 0.0400000,Welding_Angle -20.0000,Welding_CDIS 5,Welding_ACC 100,Welding_Offset {X 0.0,Y 0.0,Z 0.0}}
L270_Welding_Craft[2,5]={Welding_Name[] "S12",Welding_Pos {X 28.9999981,Y 400.000,Z -3.00000,A 0.0,B 0.0,C -23.0000},Welding_Power 80.0000,Welding_Speed 0.0400000,Welding_Angle -20.0000,Welding_CDIS 5,Welding_ACC 100,Welding_Offset {X 0.0,Y 0.0,Z 0.0}}
L270_Welding_Craft[2,6]={Welding_Name[] "S6",Welding_Pos {X 533.000,Y 463.600037,Z -2.05000,A 0.0,B -23.0000,C 0.0},Welding_Power 80.0000,Welding_Speed 0.0400000,Welding_Angle -20.0000,Welding_CDIS 5,Welding_ACC 100,Welding_Offset {X 0.0,Y 0.0,Z 0.0}}
L270_Welding_Craft[2,7]={Welding_Name[] "S7",Welding_Pos {X 533.000,Y 463.600037,Z -2.05000,A 0.0,B -23.0000,C 0.0},Welding_Power 80.0000,Welding_Speed 0.0400000,Welding_Angle -20.0000,Welding_CDIS 5,Welding_ACC 100,Welding_Offset {X 0.0,Y 0.0,Z 0.0}}
L270_Welding_Craft[2,8]={Welding_Name[] "S8",Welding_Pos {X 533.000,Y 463.600037,Z -2.05000,A 0.0,B -23.0000,C 0.0},Welding_Power 80.0000,Welding_Speed 0.0400000,Welding_Angle -20.0000,Welding_CDIS 5,Welding_ACC 100,Welding_Offset {X 0.0,Y 0.0,Z 0.0}}
L270_Welding_Craft[2,9]={Welding_Name[] "S9",Welding_Pos {X 533.000,Y 463.600037,Z -2.05000,A 0.0,B -23.0000,C 0.0},Welding_Power 80.0000,Welding_Speed 0.0400000,Welding_Angle -20.0000,Welding_CDIS 5,Welding_ACC 100,Welding_Offset {X 0.0,Y 0.0,Z 0.0}}
L270_Welding_Craft[2,10]={Welding_Name[] "S10",Welding_Pos {X 533.000,Y 338.000,Z -2.05000,A 0.0,B -23.0000,C 0.0},Welding_Power 80.0000,Welding_Speed 0.0400000,Welding_Angle -20.0000,Welding_CDIS 5,Welding_ACC 100,Welding_Offset {X 0.0,Y 0.0,Z 0.0}}

DECL GLOBAL Surr_Welding_Craft_Type C315_Welding_Craft[2,3]
C315_Welding_Craft[1,1]={Welding_Name[] "C315_S1",Welding_Pos {X 363.125,Y 660.634705,Z 1.50000,A 0.0,B 0.0,C -20.0000},Welding_Power 80.0000,Welding_Speed 0.0400000,Welding_Angle -20.0000,Welding_CDIS 5,Welding_ACC 100,Welding_Offset {X 0.0,Y -0.700000,Z -1.00000}}
C315_Welding_Craft[1,2]={Welding_Name[] "PM7",Welding_Pos {X 370.778,Y 657.395,Z 1.50000,A 0.0,B 0.0,C 0.0},Welding_Power 80.0000,Welding_Speed 0.0400000,Welding_Angle 20.0000,Welding_CDIS 5,Welding_ACC 100,Welding_Offset {X 0.0,Y 0.0,Z -1.00000},Welding_Offset_CIR {C_X 0.0,C_Y 0.0,C_Z 0.0}}
C315_Welding_Craft[1,3]={Welding_Name[] "PE7",Welding_Pos {X 375.130585,Y 648.641,Z 1.50000,A 0.0,B 20.0000,C 0.0},Welding_Power 58.0000,Welding_Speed 0.0200000,Welding_Angle 20.0000,Welding_CDIS 5,Welding_ACC 100,Welding_Offset {X -1.00000,Y -0.700000,Z -1.00000}}
C315_Welding_Craft[2,1]={Welding_Name[] "C315_S1",Welding_Pos {X 363.531,Y 661.346375,Z 1.50000,A 0.0,B 0.0,C -20.0000},Welding_Power 60.0000,Welding_Speed 0.0300000,Welding_Angle -20.0000,Welding_CDIS -1,Welding_ACC 80,Welding_Offset {X 0.0,Y -0.500000,Z -1.50000}}
C315_Welding_Craft[2,2]={Welding_Name[] "PM7",Welding_Pos {X 371.252,Y 658.128,Z 1.50000,A 0.0,B 0.0,C 0.0},Welding_Power 54.0000,Welding_Speed 0.0400000,Welding_Angle 20.0000,Welding_CDIS 5,Welding_ACC 100,Welding_Offset {X -0.300000,Y 0.0,Z 1.00000},Welding_Offset_CIR {C_X 0.0,C_Y 0.0,C_Z 0.0}}
C315_Welding_Craft[2,3]={Welding_Name[] "PE7",Welding_Pos {X 375.537689,Y 649.361,Z 1.50000,A 0.0,B 20.0000,C 0.0},Welding_Power 54.0000,Welding_Speed 0.0200000,Welding_Angle 20.0000,Welding_CDIS 5,Welding_ACC 100,Welding_Offset {X -0.100000,Y -0.100000,Z 1.00000}}


DECL GLOBAL Surr_Welding_Craft_Type N45_Short_Craft[2,5]
N45_Short_Craft[1,1]={Welding_Name[] "S5",Welding_Pos {X 364.000,Y 0.0,Z -150.000,A 0.0,B 0.0,C 0.0},Welding_Power 80.0000,Welding_Speed 0.500000,Welding_Angle 0.0,Welding_CDIS 0,Welding_ACC 100,Welding_Offset {X 0.0,Y 0.0,Z 0.0}}
N45_Short_Craft[1,2]={Welding_Name[] "S13",Welding_Pos {X 364.000,Y 0.0,Z 0.0,A 0.0,B 0.0,C 0.0},Welding_Power 80.0000,Welding_Speed 0.500000,Welding_Angle 0.0,Welding_CDIS 0,Welding_ACC 100,Welding_Offset {X 0.0,Y 0.0,Z 0.0}}
N45_Short_Craft[1,3]={Welding_Name[] "S14",Welding_Pos {X 364.000,Y 23.0000,Z 0.0,A 0.0,B 0.0,C 0.0},Welding_Power 80.0000,Welding_Speed 0.01000000,Welding_Angle 0.0,Welding_CDIS 0,Welding_ACC 100,Welding_Offset {X 0.0,Y 0.0,Z 0.0}}
N45_Short_Craft[1,4]={Welding_Name[] "S4",Welding_Pos {X 364.000,Y 20.7000,Z -150.000,A 0.0,B 0.0,C 0.0},Welding_Power 80.0000,Welding_Speed 0.500000,Welding_Angle 0.0,Welding_CDIS 0,Welding_ACC 100,Welding_Offset {X 0.0,Y 0.0,Z 0.0}}
N45_Short_Craft[1,5]={Welding_Name[] "S12",Welding_Pos {X 28.9999981,Y 400.000,Z -3.00000,A 0.0,B 0.0,C -23.0000},Welding_Power 80.0000,Welding_Speed 0.500000,Welding_Angle 0.0,Welding_CDIS 0,Welding_ACC 100,Welding_Offset {X 0.0,Y 0.0,Z 0.0}}
N45_Short_Craft[2,1]={Welding_Name[] "S5",Welding_Pos {X 362.596,Y -0.482000,Z -150.000,A 0.0,B 0.0,C 0.0},Welding_Power 80.0000,Welding_Speed 0.500000,Welding_Angle 0.0,Welding_CDIS 0,Welding_ACC 100,Welding_Offset {X 0.0,Y 0.0,Z 0.0}}
N45_Short_Craft[2,2]={Welding_Name[] "S13",Welding_Pos {X 362.596,Y -0.482000,Z 0.0,A 0.0,B 0.0,C 0.0},Welding_Power 80.0000,Welding_Speed 0.500000,Welding_Angle 0.0,Welding_CDIS 0,Welding_ACC 100,Welding_Offset {X 0.0,Y 0.0,Z 0.0}}
N45_Short_Craft[2,3]={Welding_Name[] "S14",Welding_Pos {X 362.546,Y 18.7470,Z 0.0,A 0.0,B 0.0,C 0.0},Welding_Power 80.0000,Welding_Speed 0.01000000,Welding_Angle 0.0,Welding_CDIS 0,Welding_ACC 100,Welding_Offset {X 0.0,Y 0.0,Z 0.0}}
N45_Short_Craft[2,4]={Welding_Name[] "S4",Welding_Pos {X 362.566040,Y 11.0408678,Z -150.000,A 0.0,B 0.0,C 0.0},Welding_Power 80.0000,Welding_Speed 0.500000,Welding_Angle 0.0,Welding_CDIS 0,Welding_ACC 100,Welding_Offset {X 0.0,Y 0.0,Z 0.0}}
N45_Short_Craft[2,5]={Welding_Name[] "S12",Welding_Pos {X 28.9999981,Y 400.000,Z -3.00000,A 0.0,B 0.0,C -23.0000},Welding_Power 80.0000,Welding_Speed 0.500000,Welding_Angle 0.0,Welding_CDIS 0,Welding_ACC 100,Welding_Offset {X 0.0,Y 0.0,Z 0.0}}

DECL GLOBAL Surr_Welding_Craft_Type N135_Short_Craft[2,5]
N135_Short_Craft[1,1]={Welding_Name[] "S9",Welding_Pos {X 36.0000,Y 0.0,Z -150.000,A 0.0,B 0.0,C 0.0},Welding_Power 80.0000,Welding_Speed 0.500000,Welding_Angle 0.0,Welding_CDIS 0,Welding_ACC 100,Welding_Offset {X 0.0,Y 0.0,Z 0.0}}
N135_Short_Craft[1,2]={Welding_Name[] "S13",Welding_Pos {X 36.0000,Y 0.0,Z 0.0,A 0.0,B 0.0,C 0.0},Welding_Power 80.0000,Welding_Speed 0.500000,Welding_Angle 0.0,Welding_CDIS 0,Welding_ACC 100,Welding_Offset {X 0.0,Y 0.0,Z 0.0}}
N135_Short_Craft[1,3]={Welding_Name[] "S14",Welding_Pos {X 36.0000,Y 23.0000,Z 0.0,A 0.0,B 0.0,C 0.0},Welding_Power 80.0000,Welding_Speed 0.01000000,Welding_Angle 0.0,Welding_CDIS 0,Welding_ACC 100,Welding_Offset {X 0.0,Y 0.0,Z 0.0}}
N135_Short_Craft[1,4]={Welding_Name[] "S4",Welding_Pos {X 36.0000,Y 20.7000,Z -150.000,A 0.0,B 0.0,C 0.0},Welding_Power 80.0000,Welding_Speed 0.500000,Welding_Angle 0.0,Welding_CDIS 0,Welding_ACC 100,Welding_Offset {X 0.0,Y 0.0,Z 0.0}}
N135_Short_Craft[1,5]={Welding_Name[] "S12",Welding_Pos {X 28.9999981,Y 400.000,Z -3.00000,A 0.0,B 0.0,C -23.0000},Welding_Power 80.0000,Welding_Speed 0.500000,Welding_Angle 0.0,Welding_CDIS 0,Welding_ACC 100,Welding_Offset {X 0.0,Y 0.0,Z 0.0}}
N135_Short_Craft[2,1]={Welding_Name[] "S9",Welding_Pos {X 32.1370,Y -0.736000,Z -150.000,A 0.0,B 0.0,C 0.0},Welding_Power 80.0000,Welding_Speed 0.500000,Welding_Angle 0.0,Welding_CDIS 0,Welding_ACC 100,Welding_Offset {X 0.0,Y 0.0,Z 0.0}}
N135_Short_Craft[2,2]={Welding_Name[] "S13",Welding_Pos {X 32.1370,Y -0.736000,Z 0.0,A 0.0,B 0.0,C 0.0},Welding_Power 80.0000,Welding_Speed 0.500000,Welding_Angle 0.0,Welding_CDIS 0,Welding_ACC 100,Welding_Offset {X 0.0,Y 0.0,Z 0.0}}
N135_Short_Craft[2,3]={Welding_Name[] "S14",Welding_Pos {X 32.1600,Y 18.4470,Z 0.0,A 0.0,B 0.0,C 0.0},Welding_Power 80.0000,Welding_Speed 0.01000000,Welding_Angle 0.0,Welding_CDIS 0,Welding_ACC 100,Welding_Offset {X 0.0,Y 0.0,Z 0.0}}
N135_Short_Craft[2,4]={Welding_Name[] "S4",Welding_Pos {X 32.1485,Y 8.85550117,Z -150.000,A 0.0,B 0.0,C 0.0},Welding_Power 80.0000,Welding_Speed 0.500000,Welding_Angle 0.0,Welding_CDIS 0,Welding_ACC 100,Welding_Offset {X 0.0,Y 0.0,Z 0.0}}
N135_Short_Craft[2,5]={Welding_Name[] "S12",Welding_Pos {X 28.9999981,Y 400.000,Z -3.00000,A 0.0,B 0.0,C -23.0000},Welding_Power 80.0000,Welding_Speed 0.500000,Welding_Angle 0.0,Welding_CDIS 0,Welding_ACC 100,Welding_Offset {X 0.0,Y 0.0,Z 0.0}}

DECL GLOBAL Surr_Welding_Craft_Type N225_Short_Craft[2,5]
N225_Short_Craft[1,1]={Welding_Name[] "S13",Welding_Pos {X 36.0000,Y 680.000,Z -150.000,A 0.0,B 0.0,C 0.0},Welding_Power 80.0000,Welding_Speed 0.500000,Welding_Angle 0.0,Welding_CDIS 0,Welding_ACC 100,Welding_Offset {X 0.0,Y 0.0,Z 0.0}}
N225_Short_Craft[1,2]={Welding_Name[] "S13",Welding_Pos {X 36.0000,Y 680.000,Z 0.0,A 0.0,B 0.0,C 0.0},Welding_Power 80.0000,Welding_Speed 0.500000,Welding_Angle 0.0,Welding_CDIS 0,Welding_ACC 100,Welding_Offset {X 0.0,Y 0.0,Z 0.0}}
N225_Short_Craft[1,3]={Welding_Name[] "S14",Welding_Pos {X 36.0000,Y 657.000,Z 0.0,A 0.0,B 0.0,C 0.0},Welding_Power 80.0000,Welding_Speed 0.01000000,Welding_Angle 0.0,Welding_CDIS 0,Welding_ACC 100,Welding_Offset {X 0.0,Y 0.0,Z 0.0}}
N225_Short_Craft[1,4]={Welding_Name[] "S4",Welding_Pos {X 36.0000,Y 667.500,Z -150.000,A 0.0,B 0.0,C 0.0},Welding_Power 80.0000,Welding_Speed 0.500000,Welding_Angle 0.0,Welding_CDIS 0,Welding_ACC 100,Welding_Offset {X 0.0,Y 0.0,Z 0.0}}
N225_Short_Craft[1,5]={Welding_Name[] "S12",Welding_Pos {X 28.9999981,Y 400.000,Z -3.00000,A 0.0,B 0.0,C -23.0000},Welding_Power 80.0000,Welding_Speed 0.500000,Welding_Angle 0.0,Welding_CDIS 0,Welding_ACC 100,Welding_Offset {X 0.0,Y 0.0,Z 0.0}}
N225_Short_Craft[2,1]={Welding_Name[] "S13",Welding_Pos {X 31.6630,Y 678.803,Z -150.000,A 0.0,B 0.0,C 0.0},Welding_Power 80.0000,Welding_Speed 0.500000,Welding_Angle 0.0,Welding_CDIS 0,Welding_ACC 100,Welding_Offset {X 0.0,Y 0.0,Z 0.0}}
N225_Short_Craft[2,2]={Welding_Name[] "S13",Welding_Pos {X 31.6630,Y 678.803,Z 0.0,A 0.0,B 0.0,C 0.0},Welding_Power 80.0000,Welding_Speed 0.500000,Welding_Angle 0.0,Welding_CDIS 0,Welding_ACC 100,Welding_Offset {X 0.0,Y 0.0,Z 0.0}}
N225_Short_Craft[2,3]={Welding_Name[] "S14",Welding_Pos {X 31.3610,Y 659.596,Z 0.0,A 0.0,B 0.0,C 0.0},Welding_Power 80.0000,Welding_Speed 0.01000000,Welding_Angle 0.0,Welding_CDIS 0,Welding_ACC 100,Welding_Offset {X 0.0,Y 0.0,Z 0.0}}
N225_Short_Craft[2,4]={Welding_Name[] "S4",Welding_Pos {X 31.5120010,Y 669.199463,Z -150.000,A 0.0,B 0.0,C 0.0},Welding_Power 80.0000,Welding_Speed 0.500000,Welding_Angle 0.0,Welding_CDIS 0,Welding_ACC 100,Welding_Offset {X 0.0,Y 0.0,Z 0.0}}
N225_Short_Craft[2,5]={Welding_Name[] "S12",Welding_Pos {X 28.9999981,Y 400.000,Z -3.00000,A 0.0,B 0.0,C -23.0000},Welding_Power 80.0000,Welding_Speed 0.500000,Welding_Angle 0.0,Welding_CDIS 0,Welding_ACC 100,Welding_Offset {X 0.0,Y 0.0,Z 0.0}}

DECL GLOBAL Surr_Welding_Craft_Type N315_Short_Craft[2,5]
N315_Short_Craft[1,1]={Welding_Name[] "S17",Welding_Pos {X 364.000,Y 680.000,Z -150.000,A 0.0,B 0.0,C 0.0},Welding_Power 80.0000,Welding_Speed 0.500000,Welding_Angle 0.0,Welding_CDIS 0,Welding_ACC 100,Welding_Offset {X 0.0,Y 0.0,Z 0.0}}
N315_Short_Craft[1,2]={Welding_Name[] "S13",Welding_Pos {X 364.000,Y 680.000,Z 0.0,A 0.0,B 0.0,C 0.0},Welding_Power 80.0000,Welding_Speed 0.500000,Welding_Angle 0.0,Welding_CDIS 0,Welding_ACC 100,Welding_Offset {X 0.0,Y 0.0,Z 0.0}}
N315_Short_Craft[1,3]={Welding_Name[] "S14",Welding_Pos {X 364.000,Y 657.000,Z 0.0,A 0.0,B 0.0,C 0.0},Welding_Power 80.0000,Welding_Speed 0.01000000,Welding_Angle 0.0,Welding_CDIS 0,Welding_ACC 100,Welding_Offset {X 0.0,Y 0.0,Z 0.0}}
N315_Short_Craft[1,4]={Welding_Name[] "S4",Welding_Pos {X 364.000,Y 667.500,Z -150.000,A 0.0,B 0.0,C 0.0},Welding_Power 80.0000,Welding_Speed 0.500000,Welding_Angle 0.0,Welding_CDIS 0,Welding_ACC 100,Welding_Offset {X 0.0,Y 0.0,Z 0.0}}
N315_Short_Craft[1,5]={Welding_Name[] "S12",Welding_Pos {X 28.9999981,Y 400.000,Z -3.00000,A 0.0,B 0.0,C -23.0000},Welding_Power 80.0000,Welding_Speed 0.500000,Welding_Angle 0.0,Welding_CDIS 0,Welding_ACC 100,Welding_Offset {X 0.0,Y 0.0,Z 0.0}}
N315_Short_Craft[2,1]={Welding_Name[] "S17",Welding_Pos {X 361.885,Y 679.437,Z -150.000,A 0.0,B 0.0,C 0.0},Welding_Power 80.0000,Welding_Speed 0.500000,Welding_Angle 0.0,Welding_CDIS 0,Welding_ACC 100,Welding_Offset {X 0.0,Y 0.0,Z 0.0}}
N315_Short_Craft[2,2]={Welding_Name[] "S13",Welding_Pos {X 361.885,Y 679.437,Z 0.0,A 0.0,B 0.0,C 0.0},Welding_Power 80.0000,Welding_Speed 0.500000,Welding_Angle 0.0,Welding_CDIS 0,Welding_ACC 100,Welding_Offset {X 0.0,Y 0.0,Z 0.0}}
N315_Short_Craft[2,3]={Welding_Name[] "S14",Welding_Pos {X 361.560,Y 660.457,Z 0.0,A 0.0,B 0.0,C 0.0},Welding_Power 80.0000,Welding_Speed 0.01000000,Welding_Angle 0.0,Welding_CDIS 0,Welding_ACC 100,Welding_Offset {X 0.0,Y 0.0,Z 0.0}}
N315_Short_Craft[2,4]={Welding_Name[] "S4",Welding_Pos {X 361.722504,Y 669.947,Z -150.000,A 0.0,B 0.0,C 0.0},Welding_Power 80.0000,Welding_Speed 0.500000,Welding_Angle 0.0,Welding_CDIS 0,Welding_ACC 100,Welding_Offset {X 0.0,Y 0.0,Z 0.0}}
N315_Short_Craft[2,5]={Welding_Name[] "S12",Welding_Pos {X 28.9999981,Y 400.000,Z -3.00000,A 0.0,B 0.0,C -23.0000},Welding_Power 80.0000,Welding_Speed 0.500000,Welding_Angle 0.0,Welding_CDIS 0,Welding_ACC 100,Welding_Offset {X 0.0,Y 0.0,Z 0.0}}

DECL GLOBAL E6POS Vision_Result_POS={X 175.013321,Y -792.138306,Z 222.764145,A 0.0,B 0.0,C 0.0}


DECL GLOBAL Surround_Welding_Type N1_Sink_Data={Sink_Size_Long 640.000,Sink_Size_Width 355.000,Sink_Size_R 12.0000,Sink_Size_Short_Side 20.0000,Sink_Size_Short_OnePos 31.2000,Sink_Size_Short_TwoPos 332.700,Sink_Size_Pots_Thick 0.0,Sink_Size_Panel_Thick -1.50000,Sink_Model 902182,Sink_Size_Left_Distance 20.0000,Sink_Size_Down_Distance 20.0000,Sink_Type #LeftRight_One}
DECL GLOBAL Surround_Welding_Type N2_Sink_Data={Sink_Size_Long 640.000,Sink_Size_Width 355.000,Sink_Size_R 12.0000,Sink_Size_Short_Side 20.0000,Sink_Size_Short_OnePos 31.2000,Sink_Size_Short_TwoPos 332.700,Sink_Size_Pots_Thick 0.0,Sink_Size_Panel_Thick -1.50000,Sink_Model 902182,Sink_Size_Left_Distance 20.0000,Sink_Size_Down_Distance 20.0000,Sink_Type #LeftRight_One}
;-----------Viion_INI------------



DECL GLOBAL INT Vision_Scope=20
DECL GLOBAL REAL Vision_Trans_Max_Offset=20.0000
DECL GLOBAL REAL Vision_Rota_Max_Offset=5.00000
DECL GLOBAL Vision_Type_Enum Vision_Type=#Vision_Text
;GLOBAL CHAR $Socket_Connect[1024]
;DECL GLOBAL CHAR $SOCKET_MESS[1024]
;DECL GLOBAL MODEL_TYPE $N_1
;DECL GLOBAL MODEL_TYPE $N_2
;DECL GLOBAL INT $MY_Work_Number=-1
DECL GLOBAL BOOL Vision_OFFSET_STATE=TRUE


;----------------------------------
ENDDAT
